(* IEC 61131-3 sources: CodesysTest/alpha/export/FBs/Components/FB_Funnel.pou/ClosingTime.prop, 1 file *)

(* ---- Set.pm.st ---- *)
(*#-#-#-#-#-#-#-#-#-#---Declaration---#-#-#-#-#-#-#-#-#-#-#-#-#*)

VAR
END_VAR
(*#-#-#-#-#-#-#-#-#-#---Implementation---#-#-#-#-#-#-#-#-#-#-#-#-#*)

closingTimer.PT := TO_TIME(ClosingTime * 1000);
